(* Standard MKS 909 hot cathode with gauge on reedback*)
(* works for 972 and 925 *)

FUNCTION_BLOCK FB_MKS909_RBK EXTENDS FB_GaugeBase

VAR_INPUT
    PG	: ST_VG;
END_VAR
VAR_OUTPUT
    {attribute 'pytmc' := '
    pv:
    '}
    IG	: ST_VG;
END_VAR
VAR_IN_OUT

END_VAR
VAR
    rV : REAL;
    rMaxPressure	:	REAL := 5E-2; //Torr
    rMinPressure	:	REAL := 1E-10; //Torr
    rOffPressure	:	REAL := 0.0;
    timer:TON;
    (*Default set point 50 mT*)
    rDefaultVAC_SP: REAL := 9E-3; // as per manual
    iTermBits: UINT := 30518 ; // The terminal's maximum value in bits default el3174 as per vacuum architecture
    (*IO*)
    i_iPRESS_R AT%I* :INT; // input Pressure // Link to analog Input
    q_xHV_DIS AT %Q* : BOOL := TRUE; // Active Low
    i_xGauge_ON AT %I*	: BOOL; //  True when gauge has power  // 'TcLinkTo' (EL1084) ^Input

END_VAR

(* Standard MKS 9XX series conversion *)
(* works for 972 and 925 *)

//Default setpoint 50 mT
IF PG.rVAC_SP = 0 THEN
    PG.rVAC_SP := rDefaultVAC_SP;
END_IF
// check no div by zero
If (iTermBits=0) THEN iTermBits := 30518;END_IF
rV := 10*INT_TO_REAL(IG.i_iPRESS_R)/iTermBits;

(* Pressure OK check *)
// Gauge state
// Is the gauge plugged in, and within a reasonable range?
IF i_xGauge_ON THEN
    IF  (rV >= 0.1 AND rV <=8.7) THEN // as per manual
        IG.rPRESS := LREAL_TO_REAL(EXPT(10, rV-10));
        IG.eState := Valid;
        IG.xPRESS_OK := TRUE; //Backwards compatibility
    ELSIF rV > 8.7 AND rV < 10 THEN
        IG.rPRESS :=rOffPressure;
        IG.xPRESS_OK := FALSE;
        IG.eState := Off;
    ELSE
        IG.rPRESS := rOffPressure;
        IG.xPRESS_OK := FALSE;
        IG.eState := OoR;
    END_IF
ELSE
    IG.rPRESS := rOffPressure;
    IG.xPRESS_OK := FALSE;
    IG.eState := GaugeDisconnected;
END_IF


IF (PG.rPRESS <= IG.rPRO_SP)  AND (PG.xPRESS_OK) THEN
         IG.q_xHV_DIS := IG.xHV_SW;
         IG.xILKOk := TRUE;
    ELSIF NOT IG.q_xHV_DIS AND timer.Q THEN
        IF IG.rPRESS > (IG.rPRO_SP + IG.rHYS_PR) OR PG.rPRESS > (IG.rPRO_SP + IG.rHYS_PR) THEN
        IG.q_xHV_DIS := FALSE;
        IG.xHV_SW := FALSE;
        END_IF
    ELSE
        IG.q_xHV_DIS := FALSE;
        IG.xHV_SW := FALSE;
        IG.xILKOk := FALSE;
     END_IF


timer(IN:= NOT IG.q_xHV_DIS, PT:= T#2s);

(* Setpoint evaluation *)
IG.xAT_VAC := IG.xPRESS_OK AND (IG.rPRESS < IG.rVAC_SP);

(*Soft IO Mapping*)
ACT_IO();
(*Load or save the persistent variables*)
ACT_Persistent();

(*Logger*)
THIS^.ACT_Logger();

(*Load or save the persistent variables*)
ACT_Persistent();

ACTION ACT_IO:
(*soft link inputs*)
IG.i_iPRESS_R:=	i_iPRESS_R;

(*soft link outputs*)
q_xHV_DIS := IG.q_xHV_DIS;
END_ACTION

ACTION ACT_Logger:
// ILK logger
IF NOT IG.xILKOk AND NOT IG.q_xHV_DIS THEN
         fbLogger(sMsg:='Lost external interlock while gauge was on.', eSevr:=TcEventSeverity.Critical);
END_IF


// Log Action
tAction(CLK:=  IG.q_xHV_DIS);
IF tAction.Q THEN fbLogger(sMsg:='Ion gauge commanded to switch on', eSevr:=TcEventSeverity.Info); END_IF



//STATE Logger
IF ePrevState <> IG.eState THEN
      CASE IG.eState OF
        ValidHi:
        ValidLo:
        Valid:
            fbLogger(sMsg:='Gauge pressure valid.', eSevr:=TcEventSeverity.Info);
          GaugeDisconnected:
            fbLogger(sMsg:='Gauge Disconnected.', eSevr:=TcEventSeverity.Critical);
        PressInvalid:
            fbLogger(sMsg:='Gauge pressure invalid.', eSevr:=TcEventSeverity.Warning);
        OoR:
            fbLogger(sMsg:='Gauge pressure out of range.', eSevr:=TcEventSeverity.Warning);
        Starting:
            fbLogger(sMsg:='Gauge starting.', eSevr:=TcEventSeverity.Info);
      END_CASE
      ePrevState := IG.eState;
END_IF
END_ACTION

ACTION ACT_Persistent:
(*On first PLC pass, load the persistent value into the structrue variable*)
IF (SUPER^.bRestorePersistentData) THEN
    SUPER^.bRestorePersistentData	:= FALSE;
    IF ( rVAC_SP <> 0) THEN
        IG.rVAC_SP := rVAC_SP;
    END_IF;
    IF ( rPRO_SP <> 0) THEN
        IG.rPRO_SP := rPRO_SP;
    END_IF;
    IF ( rHYS_PR <> 0) THEN
        IG.rHYS_PR := rHYS_PR;
    END_IF;
END_IF
(*Check if a new value has been written in the structure variable copy it to the persistent variable*)
IF NOT (IG.rVAC_SP = rVAC_SP)  THEN
    rVAC_SP := IG.rVAC_SP;
END_IF;

IF NOT (IG.rPRO_SP = rPRO_SP) THEN
    rPRO_SP:= IG.rPRO_SP;
END_IF;

IF NOT (IG.rHYS_PR = rHYS_PR) THEN
    rHYS_PR:= IG.rHYS_PR;
END_IF;
END_ACTION

METHOD M_AutoOn : BOOL
VAR_INPUT
END_VAR
this^.IG.q_xHV_DIS:= FALSE;
END_METHOD

METHOD M_SetBits : BOOL
VAR_INPUT
    TermBits : UINT; // The terminal's maximum value in bits
END_VAR
This^.iTermBits := TermBits;
END_METHOD

END_FUNCTION_BLOCK

(* stored: Version 1.1.0.1
   POU FB_MKS909_RBK: Id {e4d3e807-daeb-4a47-bccf-64bd129edfcd}, SpecialFunc None
   Action ACT_IO: Id {89c7028d-3190-45b7-aaec-73bdcb00e265}
   Action ACT_Logger: Id {c289ef5c-0d6d-44e6-b87e-b28bbd141dbf}
   Action ACT_Persistent: Id {ba42c9e0-fb4b-4426-98a9-0712e0f03714}
   Method M_AutoOn: Id {6fde0073-91f6-4cb9-bbee-4ff5715804d3}
   Method M_SetBits: Id {a0b5c519-56d7-42f9-be00-fe9985112627} *)
